FUNCTION_BLOCK FB_BoxLED IMPLEMENTS ITF_SubSystem
VAR_INPUT
	eMode : LEDMode;
END_VAR
VAR
	//Local
	iBoxLED : INT;
	fbFlashingTimer : TON;
	bOn : BOOL;
	
	//ErrorBits
	bTemperatureTooHigh : BIT;
	bNoSupplyVoltage : BIT;
END_VAR
VAR CONSTANT
	iIntensity : INT := 32767;				//Intensity [0..32767]
	rDimFactor : REAL := 0.01;				//Percentage (0..100%)
	tSlowFlashingTime : TIME := T#1S;		
	tFastFlashingTime : TIME := T#100MS;
END_VAR

CASE eMode OF
	LEDMode.Off:
			doTurnOn(iBrightness := 0);
	LEDMode.On:
			doTurnOn(iBrightness := iIntensity);
	LEDMode.Dimmed:
			doDimming(rDimmingFactor:=rDimFactor);
	LEDMode.SlowFlashing:
			doFlashing(FlashingTime:=tSlowFlashingTime);
	LEDMode.FastFlashing:
			doFlashing(FlashingTime:=tFastFlashingTime);
END_CASE

doSetClampValues();
doGetClampValues();

METHOD PRIVATE doDimming
VAR_INPUT
	rDimmingFactor : REAL;
END_VAR
iBoxLED := REAL_TO_INT(rDimmingFactor * iIntensity);
END_METHOD

METHOD PRIVATE doFlashing
VAR_INPUT
	FlashingTime : TIME;
END_VAR
fbFlashingTimer(IN:=TRUE, PT:=FlashingTime);
IF fbFlashingTimer.Q THEN
	fbFlashingTimer(IN:=FALSE);
	bOn := NOT bOn;	
END_IF
IF bOn THEN
	iBoxLED := iIntensity;
ELSE
	iBoxLED := 0;
END_IF
END_METHOD

METHOD PRIVATE doGetClampValues
bTemperatureTooHigh := BoxLED.bWhiteWarning;
bNoSupplyVoltage := BoxLED.bWhiteError;
END_METHOD

METHOD PRIVATE doSetClampValues
BoxLED.iWhite := iBoxLED;
END_METHOD

METHOD PRIVATE doTurnOn
VAR_INPUT
	iBrightness : INT;
END_VAR
iBoxLED := iBrightness;
END_METHOD

PROPERTY eCondition : SubLevelCondition
GET
IF nErrorID <> 0 THEN
	eCondition := SubLevelCondition.ERROR;
ELSE
	eCondition := SubLevelCondition.RUN;
END_IF
END_GET
END_PROPERTY

PROPERTY nErrorID : UDINT
GET
nErrorID.0 := bTemperatureTooHigh;
nErrorID.1 := bNoSupplyVoltage;
END_GET
END_PROPERTY

END_FUNCTION_BLOCK

(* stored: Version 1.1.0.1, ProductVersion 3.1.4024.12
   POU FB_BoxLED: Id {7417f049-9846-439d-bd3a-1b6848121830}, SpecialFunc None
   Method doDimming: Id {ef13b277-d6e0-4180-8bd3-5ca9a77d8ba4}
   Method doFlashing: Id {a56a3bcf-ecb7-4bdc-afc1-de57457e0ffa}
   Method doGetClampValues: Id {ed091663-cac3-4e07-8db6-bc90a174ab60}
   Method doSetClampValues: Id {dc51a952-fa37-42fa-8053-b84e73c61317}
   Method doTurnOn: Id {ff9f7808-2e93-4ad9-ae70-22394be7f716}
   Property eCondition: Id {4e482d49-3544-41a4-af6c-918dcc95d53c}
   Get Get: Id {79825f0a-16ce-4375-9182-20617a9508fb}
   Property nErrorID: Id {5e4b59cd-ff12-43ce-a556-f3f12e731d20}
   Get Get: Id {3a0b74a6-2860-46c3-baf9-490027dc347b} *)
